ABB RobotStudio station: Project7_1.rsstnx

Station Project7 (saved by RobotStudio 22.3.10190.2)
Layout (positions relative to the parent item):
  - Gorionik [mechanism] at (944.87, 0, 1229) mm, rotated rx 180 ry 60 rz 180 deg
      TCP Gorionik at (0, 0, 172) mm
      links: Gorionik1
  - IRB1660ID_6_155__03 [mechanism, from Robots\IRB1660ID_6_155__03.rslib] at (0, 0, 0) mm; joint values [0, 0, 0, 0, 0.5236, 0] (rad or m)
Attachment: Gorionik is attached to IRB1660ID_6_155__03 / Link6
Targets, tools, work objects and paths stored in the station, written as RAPID:
! task (no controller)
MODULE CalibData
  PERS tooldata Gorionik:=[TRUE,[[0,0,172],[1,0,0,0]],[0.5,[0,0.113,32.05],[1,0,0,0],0,0,0]];
ENDMODULE

